FUNCTION_BLOCK FIFO_UINT (* A FIFO queue of UINTs *)
  (* Standard: 61499-1 *)
  (* Version 0.0, 2005-12-09, JHC, Holobloc Inc., Derived from STACK_INT. *)
  (* Compiler header: package fb.rt.student; *)
  (* Compiler Java Sun JDK 1.5 *)
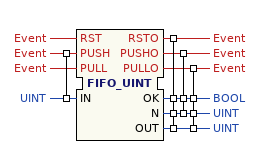
  EVENT_INPUT
    RST; (* Empty the queue *)
    PUSH WITH IN; (* Push the value of IN to the end of the queue if possible. *)
    PULL; (* Pull the value of OUT from the front of the queue if possible. *)
  END_EVENT
  EVENT_OUTPUT
    RSTO WITH N, OK, OUT; (* Reset confirmation *)
    PUSHO WITH N, OK; (* PUSH confirmation *)
    PULLO WITH OK, OUT, N; (* PULL confirmation *)
  END_EVENT
  VAR_INPUT
    IN : UINT; (* Input to be pushed *)
  END_VAR
  VAR_OUTPUT
    OK : BOOL; (* OUT value valid *)
    N : UINT; (* Number of elements in queue *)
    OUT : UINT; (* Data from last PULL - meaningless if OK = FALSE *)
  END_VAR
  VAR
    BUF : ARRAY [0..127] OF UINT; (* Circular buffer *)
    PTR : UINT; (* Location for next PUSH *)
    OUTPTR : UINT; (* Location for next PULL *)
  END_VAR
  ALGORITHM PUSH IN ST:
IF N = 128 THEN
OK := FALSE;
ELSE
OK := TRUE;
BUF[PTR] := IN;
PTR := (PTR+1)%128;
N := N+1;
END_IF;
PUSHO.serviceEvent(this);
  END_ALGORITHM
  ALGORITHM PULL IN ST:
IF N = 0 THEN
OK := FALSE;
ELSE
OK := TRUE;
OUT := BUF[OUTPTR];
OUTPTR := (OUTPTR+1)%128;
N := N-1;
END_IF;
PULLO.serviceEvent(this);
  END_ALGORITHM
  ALGORITHM RST IN ST:
PTR := 0;
OUTPTR := 0;
N := 0;
OUT := 0;
OK := FALSE;
RSTO.serviceEvent(this);
  END_ALGORITHM
END_FUNCTION_BLOCK
